SUBAPPLICATION Uebung_049 (* DigitalInput_I1-_I4 auf DigitalOutput_Q1-_Q4 *)
  (* Standard: 61499-2 *)
  (* Version 1.0, 2023-10-23, franz *)
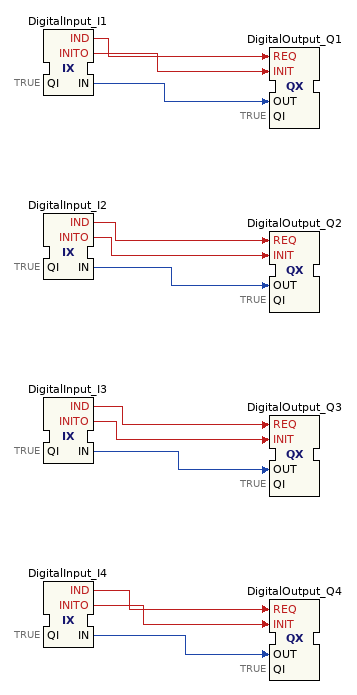
  FBS
    DigitalOutput_Q1 : QX(QI := TRUE);
    DigitalInput_I1 : IX(QI := TRUE);
    DigitalOutput_Q2 : QX(QI := TRUE);
    DigitalInput_I2 : IX(QI := TRUE);
    DigitalOutput_Q3 : QX(QI := TRUE);
    DigitalInput_I3 : IX(QI := TRUE);
    DigitalOutput_Q4 : QX(QI := TRUE);
    DigitalInput_I4 : IX(QI := TRUE);
  END_FBS
  EVENT_CONNECTIONS
    DigitalInput_I1.IND TO DigitalOutput_Q1.REQ;
    DigitalInput_I2.IND TO DigitalOutput_Q2.REQ;
    DigitalInput_I3.IND TO DigitalOutput_Q3.REQ;
    DigitalInput_I4.IND TO DigitalOutput_Q4.REQ;
    DigitalInput_I3.INITO TO DigitalOutput_Q3.INIT;
    DigitalInput_I4.INITO TO DigitalOutput_Q4.INIT;
    DigitalInput_I2.INITO TO DigitalOutput_Q2.INIT;
    DigitalInput_I1.INITO TO DigitalOutput_Q1.INIT;
  END_CONNECTIONS
  DATA_CONNECTIONS
    DigitalInput_I1.IN TO DigitalOutput_Q1.OUT;
    DigitalInput_I2.IN TO DigitalOutput_Q2.OUT;
    DigitalInput_I3.IN TO DigitalOutput_Q3.OUT;
    DigitalInput_I4.IN TO DigitalOutput_Q4.OUT;
  END_CONNECTIONS
END_SUBAPPLICATION
